// TIA Portal V17 export
// export: Created 2023-12-22T15:08:06.9150171Z, ExportSetting WithDefaults, DisplayName Totally Integrated Automation Portal, DisplayVersion V17, DisplayName TIA Portal Openness, DisplayVersion V17, DisplayName TIA Portal Version Control Interface, DisplayVersion V17, DisplayName STEP 7 Professional, DisplayVersion V17, DisplayName STEP 7 Safety, DisplayVersion V17, DisplayName WinCC Advanced, DisplayVersion V17
FUNCTION "FC_DRV_End" : Void   // FC101, LAD
{ S7_Optimized_Access := 'FALSE' }
VERSION : 0.1
// stored: AutoNumber false, IsIECCheckEnabled false, SetENOAutomatically false, UDAEnableTagReadback false
   VAR_TEMP
      ev : Bool;
   END_VAR
   VAR_TEMP   // added for the SCL form of the ladder/FBD networks
      _w1 : Bool;
      _w2 : Bool;
      _w3 : Bool;
      _w4 : Bool;
      _w5 : Bool;
      _w6 : Bool;
      _w7 : Bool;
      _w8 : Bool;
   END_VAR
BEGIN

REGION Network 1: Одно из устройств нижнего уровня в ручном режиме
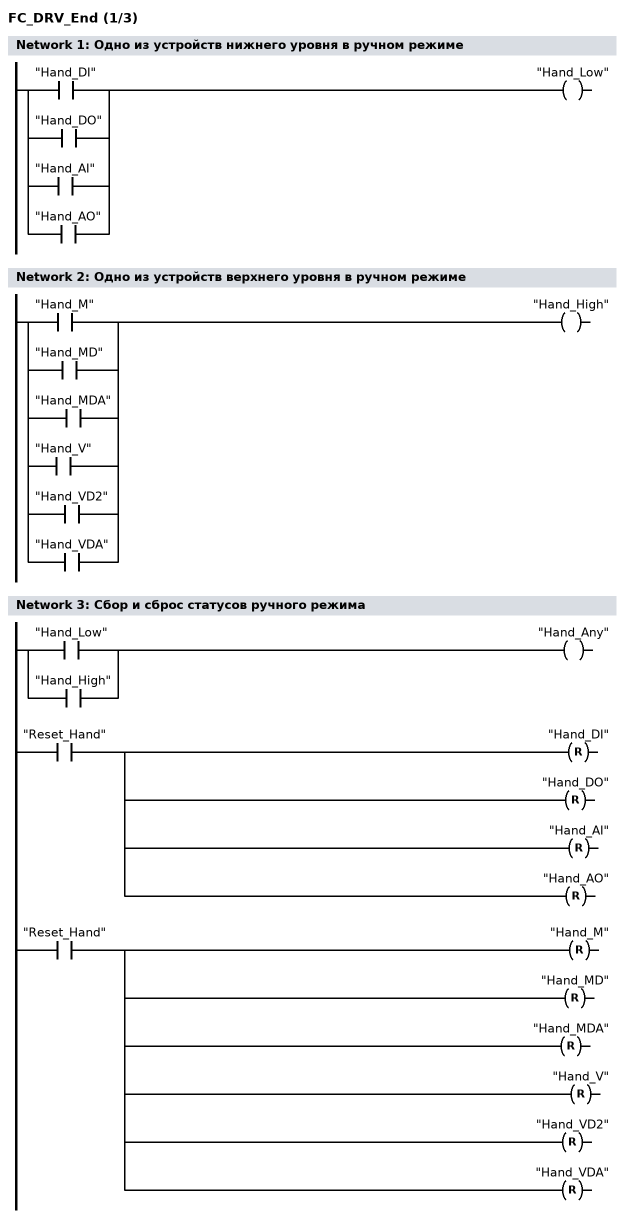
   RUNG wire#powerrail
      Contact( "Hand_DI" )
      wire#w1
      Coil( "Hand_Low" )
   END_RUNG
   RUNG wire#powerrail
      Contact( "Hand_DO" )
   END_RUNG wire#w1
   RUNG wire#powerrail
      Contact( "Hand_AI" )
   END_RUNG wire#w1
   RUNG wire#powerrail
      Contact( "Hand_AO" )
   END_RUNG wire#w1
   // the same network as SCL:
   "Hand_Low" := "Hand_DI" OR "Hand_DO" OR "Hand_AI" OR "Hand_AO";
END_REGION

REGION Network 2: Одно из устройств верхнего уровня в ручном режиме
   RUNG wire#powerrail
      Contact( "Hand_M" )
      wire#w1
      Coil( "Hand_High" )
   END_RUNG
   RUNG wire#powerrail
      Contact( "Hand_MD" )
   END_RUNG wire#w1
   RUNG wire#powerrail
      Contact( "Hand_MDA" )
   END_RUNG wire#w1
   RUNG wire#powerrail
      Contact( "Hand_V" )
   END_RUNG wire#w1
   RUNG wire#powerrail
      Contact( "Hand_VD2" )
   END_RUNG wire#w1
   RUNG wire#powerrail
      Contact( "Hand_VDA" )
   END_RUNG wire#w1
   // the same network as SCL:
   "Hand_High" := "Hand_M" OR "Hand_MD" OR "Hand_MDA" OR "Hand_V" OR "Hand_VD2" OR "Hand_VDA";
END_REGION

REGION Network 3: Сбор и сброс статусов ручного режима
   RUNG wire#powerrail
      Contact( "Hand_Low" )
      wire#w1
      Coil( "Hand_Any" )
   END_RUNG
   RUNG wire#powerrail
      Contact( "Hand_High" )
   END_RUNG wire#w1
   RUNG wire#powerrail
      Contact( "Reset_Hand" )
      wire#w2
      R_Coil( "Hand_DI" )
   END_RUNG
   RUNG wire#w2
      R_Coil( "Hand_DO" )
   END_RUNG
   RUNG wire#w2
      R_Coil( "Hand_AI" )
   END_RUNG
   RUNG wire#w2
      R_Coil( "Hand_AO" )
   END_RUNG
   RUNG wire#powerrail
      Contact( "Reset_Hand" )
      wire#w3
      R_Coil( "Hand_M" )
   END_RUNG
   RUNG wire#w3
      R_Coil( "Hand_MD" )
   END_RUNG
   RUNG wire#w3
      R_Coil( "Hand_MDA" )
   END_RUNG
   RUNG wire#w3
      R_Coil( "Hand_V" )
   END_RUNG
   RUNG wire#w3
      R_Coil( "Hand_VD2" )
   END_RUNG
   RUNG wire#w3
      R_Coil( "Hand_VDA" )
   END_RUNG
   // the same network as SCL:
   "Hand_Any" := "Hand_Low" OR "Hand_High";
   IF "Reset_Hand" THEN
       "Hand_DI" := FALSE;
       "Hand_DO" := FALSE;
       "Hand_AI" := FALSE;
       "Hand_AO" := FALSE;
       "Hand_M" := FALSE;
       "Hand_MD" := FALSE;
       "Hand_MDA" := FALSE;
       "Hand_V" := FALSE;
       "Hand_VD2" := FALSE;
       "Hand_VDA" := FALSE;
   END_IF;
END_REGION

REGION Network 4
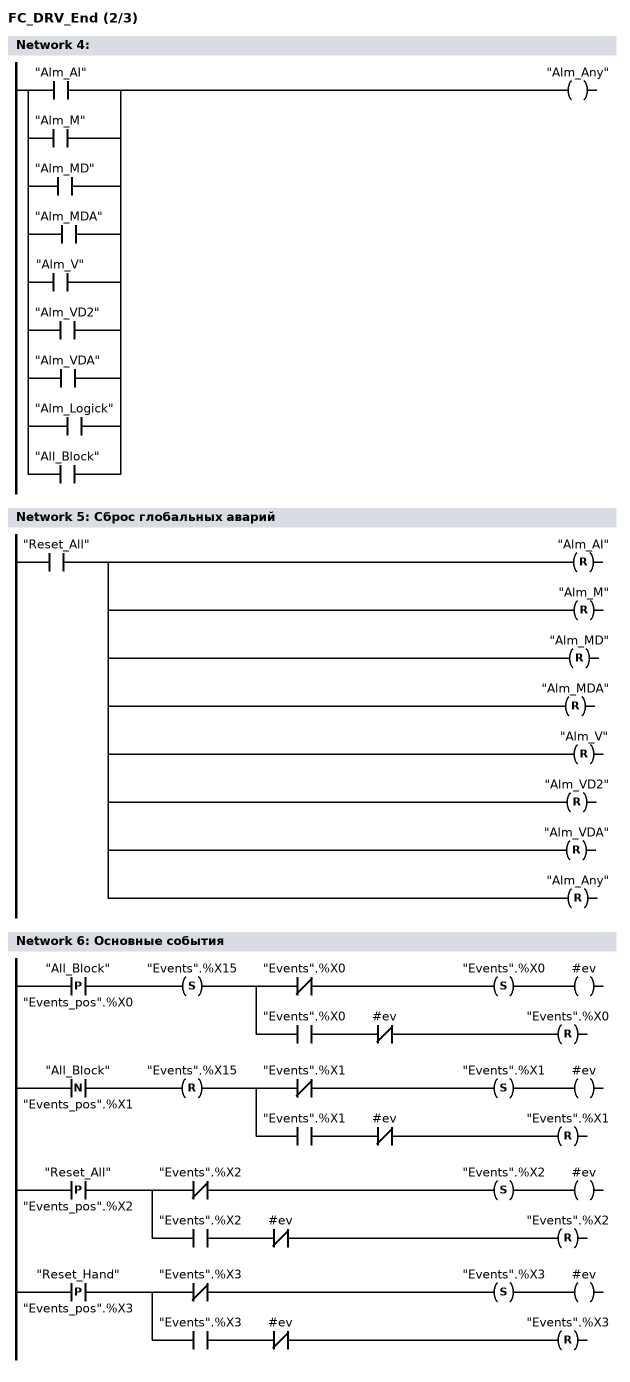
   RUNG wire#powerrail
      Contact( "Alm_AI" )
      wire#w1
      Coil( "Alm_Any" )
   END_RUNG
   RUNG wire#powerrail
      Contact( "Alm_M" )
   END_RUNG wire#w1
   RUNG wire#powerrail
      Contact( "Alm_MD" )
   END_RUNG wire#w1
   RUNG wire#powerrail
      Contact( "Alm_MDA" )
   END_RUNG wire#w1
   RUNG wire#powerrail
      Contact( "Alm_V" )
   END_RUNG wire#w1
   RUNG wire#powerrail
      Contact( "Alm_VD2" )
   END_RUNG wire#w1
   RUNG wire#powerrail
      Contact( "Alm_VDA" )
   END_RUNG wire#w1
   RUNG wire#powerrail
      Contact( "Alm_Logick" )
   END_RUNG wire#w1
   RUNG wire#powerrail
      Contact( "All_Block" )
   END_RUNG wire#w1
   // the same network as SCL:
   "Alm_Any" := "Alm_AI" OR "Alm_M" OR "Alm_MD" OR "Alm_MDA" OR "Alm_V" OR "Alm_VD2" OR "Alm_VDA" OR "Alm_Logick" OR "All_Block";
END_REGION

REGION Network 5: Сброс глобальных аварий
   RUNG wire#powerrail
      Contact( "Reset_All" )
      wire#w1
      R_Coil( "Alm_AI" )
   END_RUNG
   RUNG wire#w1
      R_Coil( "Alm_M" )
   END_RUNG
   RUNG wire#w1
      R_Coil( "Alm_MD" )
   END_RUNG
   RUNG wire#w1
      R_Coil( "Alm_MDA" )
   END_RUNG
   RUNG wire#w1
      R_Coil( "Alm_V" )
   END_RUNG
   RUNG wire#w1
      R_Coil( "Alm_VD2" )
   END_RUNG
   RUNG wire#w1
      R_Coil( "Alm_VDA" )
   END_RUNG
   RUNG wire#w1
      R_Coil( "Alm_Any" )
   END_RUNG
   // the same network as SCL:
   IF "Reset_All" THEN
       "Alm_AI" := FALSE;
       "Alm_M" := FALSE;
       "Alm_MD" := FALSE;
       "Alm_MDA" := FALSE;
       "Alm_V" := FALSE;
       "Alm_VD2" := FALSE;
       "Alm_VDA" := FALSE;
       "Alm_Any" := FALSE;
   END_IF;
END_REGION

REGION Network 6: Основные события
   RUNG wire#powerrail
      P_Contact(operand := "All_Block", bit := "Events_pos".%X0)
      S_Coil( "Events".%X15 )
      wire#w1
      I_Contact( "Events".%X0 )
      S_Coil( "Events".%X0 )
      Coil( #ev )
   END_RUNG
   RUNG wire#w1
      Contact( "Events".%X0 )
      I_Contact( #ev )
      R_Coil( "Events".%X0 )
   END_RUNG
   RUNG wire#powerrail
      N_Contact(operand := "All_Block", bit := "Events_pos".%X1)
      R_Coil( "Events".%X15 )
      wire#w2
      I_Contact( "Events".%X1 )
      S_Coil( "Events".%X1 )
      Coil( #ev )
   END_RUNG
   RUNG wire#w2
      Contact( "Events".%X1 )
      I_Contact( #ev )
      R_Coil( "Events".%X1 )
   END_RUNG
   RUNG wire#powerrail
      P_Contact(operand := "Reset_All", bit := "Events_pos".%X2)
      wire#w3
      I_Contact( "Events".%X2 )
      S_Coil( "Events".%X2 )
      Coil( #ev )
   END_RUNG
   RUNG wire#w3
      Contact( "Events".%X2 )
      I_Contact( #ev )
      R_Coil( "Events".%X2 )
   END_RUNG
   RUNG wire#powerrail
      P_Contact(operand := "Reset_Hand", bit := "Events_pos".%X3)
      wire#w4
      I_Contact( "Events".%X3 )
      S_Coil( "Events".%X3 )
      Coil( #ev )
   END_RUNG
   RUNG wire#w4
      Contact( "Events".%X3 )
      I_Contact( #ev )
      R_Coil( "Events".%X3 )
   END_RUNG
   // the same network as SCL:
   #_w1 := "All_Block" AND NOT "Events_pos".%X0;   // rising edge of "All_Block"
   "Events_pos".%X0 := "All_Block";
   IF #_w1 THEN "Events".%X15 := TRUE; END_IF;
   #_w2 := #_w1 AND NOT "Events".%X0;
   IF #_w2 THEN "Events".%X0 := TRUE; END_IF;
   #ev := #_w2;
   IF #_w1 AND "Events".%X0 AND NOT #ev THEN "Events".%X0 := FALSE; END_IF;
   #_w3 := NOT "All_Block" AND "Events_pos".%X1;   // falling edge of "All_Block"
   "Events_pos".%X1 := "All_Block";
   IF #_w3 THEN "Events".%X15 := FALSE; END_IF;
   #_w4 := #_w3 AND NOT "Events".%X1;
   IF #_w4 THEN "Events".%X1 := TRUE; END_IF;
   #ev := #_w4;
   IF #_w3 AND "Events".%X1 AND NOT #ev THEN "Events".%X1 := FALSE; END_IF;
   #_w5 := "Reset_All" AND NOT "Events_pos".%X2;   // rising edge of "Reset_All"
   "Events_pos".%X2 := "Reset_All";
   #_w6 := #_w5 AND NOT "Events".%X2;
   IF #_w6 THEN "Events".%X2 := TRUE; END_IF;
   #ev := #_w6;
   IF #_w5 AND "Events".%X2 AND NOT #ev THEN "Events".%X2 := FALSE; END_IF;
   #_w7 := "Reset_Hand" AND NOT "Events_pos".%X3;   // rising edge of "Reset_Hand"
   "Events_pos".%X3 := "Reset_Hand";
   #_w8 := #_w7 AND NOT "Events".%X3;
   IF #_w8 THEN "Events".%X3 := TRUE; END_IF;
   #ev := #_w8;
   IF #_w7 AND "Events".%X3 AND NOT #ev THEN "Events".%X3 := FALSE; END_IF;
END_REGION

REGION Network 7: Очистка DTR
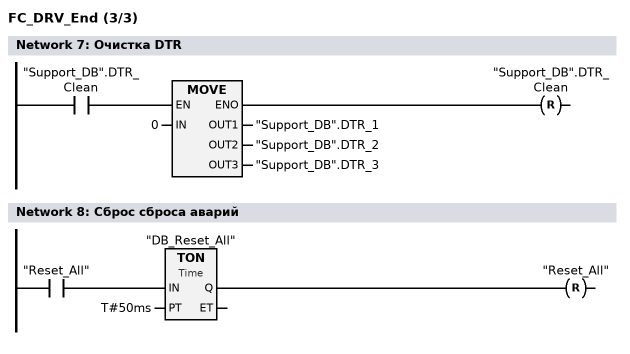
   RUNG wire#powerrail
      Contact( "Support_DB".DTR_Clean )
      Move(in := 0, out1 => "Support_DB".DTR_1, out2 => "Support_DB".DTR_2, out3 => "Support_DB".DTR_3)
      R_Coil( "Support_DB".DTR_Clean )
   END_RUNG
   // the same network as SCL:
   IF "Support_DB".DTR_Clean THEN
       "Support_DB".DTR_1 := 0;
       "Support_DB".DTR_2 := 0;
       "Support_DB".DTR_3 := 0;
       "Support_DB".DTR_Clean := FALSE;
   END_IF;
END_REGION

REGION Network 8: Сброс сброса аварий
   RUNG wire#powerrail
      Contact( "Reset_All" )
      { S7_Templates := "time_type := Time" } "DB_Reset_All".TON(pt := T#50ms, et =>)
      R_Coil( "Reset_All" )
   END_RUNG
   // the same network as SCL:
   "DB_Reset_All".TON(IN := "Reset_All", PT := T#50ms);
   IF "DB_Reset_All".Q THEN "Reset_All" := FALSE; END_IF;
END_REGION
END_FUNCTION
